(* PLC project , CODESYS CODESYS V3.5 SP16 Patch 4 *)
(* stored: creationDateTime 2021-05-19T12:12:31.4539395, modificationDateTime 2021-05-19T11:50:23.9006141 *)

FUNCTION_BLOCK baseChoiseTest_FB_anon EXTENDS FB_TestSuite

            TC1();
          

METHOD TC1
  VAR_INPUT
    t_var1 : WORD := 0;
    t_var2 : WORD := 0;
  END_VAR
  VAR
    Fun : FB_anon;
    Result_out_SetOk : BOOL;
    t_out_No2 : WORD;
    ExpectedResult : BOOL := FALSE;
    Condition : BOOL;
  END_VAR
                  TEST('TC1');	(* Naming the test case *)

(* Calling the FB to be tested *)
Fun(in_var1 := t_var1, in_var2 := t_var2, out_SetOk => Result_out_SetOk, out_No2 => t_out_No2);

AssertTrue(Condition := (Result_out_SetOk = ExpectedResult),
			Message := 'Result_out_SetOk is True');
			
TEST_FINISHED();
                
END_METHOD
END_FUNCTION_BLOCK
